FUNCTION_BLOCK MC_SYNCHRONIZEDMOTIONSIMULATION

VAR_IN_OUT
	Slave	: AXIS_REF;	(* B *)
END_VAR


VAR_INPUT


	Enable : BOOL;

END_VAR
VAR_OUTPUT

	InSimulation	:BOOL;

Busy	:BOOL;

	Error	:BOOL;

ErrorId	:WORD;

END_VAR
VAR
END_VAR

;

END_FUNCTION_BLOCK

(* stored: Version 1.1.0.1
   POU MC_SYNCHRONIZEDMOTIONSIMULATION: Id {87beaf09-5f58-4e05-893d-0a3efd88253d}, SpecialFunc None *)
